Staubli VAL3: POINT.pjx

--- POINT.pjx ---
Parameters version=s7.6.1 stackSize=5000 millimeterUnit=true
Program file=copy_it.pgx
Program file=link_all.pgx
Program file=link_it.pgx
Data file=POINT.dtx
Library alias=saveData path=Disk://saveData/SAVEDATA.pjx
Type name=TrajPoint path=Disk://kernel/template/TrajPoint/TrajPoint.pjx
Type name=FrameItem path=Disk://kernel/template/FrameItem/FrameItem.pjx

--- POINT.dtx ---
public TrajPoint tTraj{}

--- copy_it.pgx ---
public program copy_it(string x_sCopy, string x_sPaste)
  local num i
begin
  // try to copy it
  if isDefined(tTraj[x_sCopy])
    // copy it
    tTraj[x_sPaste]=tTraj[x_sCopy]
    //
  endIf
end
